TYPE ST_MESSAGE_CTRL :
STRUCT
  Cmd         : E_MESSAGE_CTRL;
END_STRUCT
END_TYPE

(* stored: Version 1.1.0.1, ProductVersion 3.1.4026.18
   DUT ST_MESSAGE_CTRL: Id {caf7b10e-42bf-40ec-bdeb-f449ce7e14bb} *)
